(* PLC project canplc, CODESYS STW CODESYS V3.5 SP11 - ESX-3CS *)
(* stored: creationDateTime 2026-05-19T11:32:05.4310643, version 0.101, modificationDateTime 2026-02-01T07:40:15, organization Isoloader *)

TYPE t_can_errorfield : ARRAY[0..5] OF WORD;
END_TYPE

TYPE t_can_heartbeaterrors : ARRAY[0..7] OF BYTE;
END_TYPE

TYPE t_canopen_emcy : CIA405.EMCY_ERROR;
END_TYPE

TYPE t_node_state : _3SCOS.DEVICE_STATE;
END_TYPE

VAR_GLOBAL  (* GlobalVariablesCanplc *)
  gCANPLCBoolA : BOOL := TRUE;
END_VAR

FUNCTION_BLOCK CANOpenLocalDevice EXTENDS OperationalParticleSet
  VAR CONSTANT
    cHeartbeatTimer : t_time := TIME#500ms;
  END_VAR
  VAR
    lAlarmCANOpenMasterNotOperational : ReportableAlarmEscalating;
    lAlarmCANOpenMasterModulation : ReportableSignedModulation;
    lAlarmCANOpenMasterAllowableUp : ReportableAlarmAllowableUp;
    lVREnabled : ValueReferenceBool;
    lEnabled : BOOL := TRUE;
    lVRTriggerStart : ValueReferenceBool;
    lTriggerStart : BOOL := FALSE;
    lVROverrideConnected : ValueReferenceBool;
    lOverrideConnected : BOOL := FALSE;
    lModulationSystemStateScope : t_system_state;
    lOperationalSystemStateScope : t_system_state;
    lStartSystemStateScope : t_system_state;
    lModulationSeverity : t_severity;
    lNetworkId : BYTE;
    _EmergencyInfo : t_canopen_emcy;  (* foobar emcy messages not monitored *)
    lEmergencyInfo : REFERENCE TO t_canopen_emcy := _EmergencyInfo;
    lControllerId : BYTE := 0;
    lCANOpenDevice : REFERENCE TO _3SCSS.CANopenDevice;
    lMasterHeartbeat : HeartbeatHandler;
    lNodeState : t_node_state;
    lNodeStatePrev : t_node_state;
    lNMTStartCounter : USINT := 0;
    lNMTTimer : t_timer;
    lNMTEnableStart : BOOL := TRUE;
    lHeartbeatCounter : Counter;
    lHeartbeatTimer : t_timer;
    lEmergencyCounter : Counter;
    lReceiveEmcy : CIA405.RECV_EMCY_DEV;
    lEmergencyCode : WORD;
    lOverflowCounter : USINT := 0;
    lConnected : BOOL := TRUE;
  END_VAR

            ;
          

METHOD initialize
                  IF (NOT(__ISVALIDREF(lCANOpenDevice))) THEN
	gCodeErrorHandler(pMessage:=CONCAT('null reference in ',lIdentity));
END_IF

lAlarmCANOpenMasterNotOperational.initializeState(NopSelf,'',cACCANOpenMasterNotOperational);
lAlarmCANOpenMasterNotOperational.InitialSeverity := cSeverityWarning;
lAlarmCANOpenMasterNotOperational.SeverityWarningTimeout := T#0S;
lAlarmCANOpenMasterNotOperational.SeverityErrorTimeout := T#100MS;
lAlarmCANOpenMasterNotOperational.SeverityCriticalTimeout := T#5S;

lAlarmCANOpenMasterModulation.initializeState(NopSelf,'',cACCANOpenMasterModulation);
lAlarmCANOpenMasterModulation.pause(); // foobar - what impact does this have, should act as if not connected, ie put all joysticks to zero

lAlarmCANOpenMasterAllowableUp.initializeState(NopSelf,'',cACCANOpenMasterAllowableUp);
lAlarmCANOpenMasterAllowableUp.AllowableSystemState := cSystemStatePreOperational;
lAlarmCANOpenMasterAllowableUp.UpperSystemStateScope := cSystemStatePreOperational;
lAlarmCANOpenMasterAllowableUp.LowerSystemStateScope := cSystemStatePreOperational;
lAlarmCANOpenMasterAllowableUp.Life := 10;
lAlarmCANOpenMasterAllowableUp.InitialSeverity := cSeverityNone;
lAlarmCANOpenMasterAllowableUp.SeverityWarningTimeout := T#250MS;
lAlarmCANOpenMasterAllowableUp.SeverityErrorTimeout := T#1S;
lAlarmCANOpenMasterAllowableUp.SeverityCriticalTimeout := T#5S;	

lVREnabled.initializeValueReference(lEnabled,NopSelf,'Enabled','Enable canopen node','',cValueStyleParameter);
lVRTriggerStart.initializeValueReference(lTriggerStart,NopSelf,'TriggerStart','Trigger NMT message to take canopen node Operational','',cValueStyleTrigger);
lVROverrideConnected.initializeValueReference(lOverrideConnected,NopSelf,'OvrdConnected','Force state of canopen node to show as connected','',cValueStyleParameter);

SUPER^.initialize();
	
lModulationSystemStateScope := cSystemStateOperational;	
lOperationalSystemStateScope := cSystemStateGoOperational;
lStartSystemStateScope := cSystemStateGoOperational;
lModulationSeverity := cSeverityError;

lHeartbeatCounter.initialize();
lEmergencyCounter.initialize();
lMasterHeartbeat.initialize();

lHeartbeatTimer.initialize();
lHeartbeatTimer.Enable := TRUE;
lHeartbeatTimer.Period := cHeartbeatTimer;

lControllerId := lCANOpenDevice.NodeID;

lNMTStartCounter := 0;
lNMTTimer.Enable := TRUE;
lNMTTimer.Period := T#250MS;


                
END_METHOD

METHOD start
                  lCANOpenDevice.SwitchToOp();

lNMTStartCounter := lNMTStartCounter + 1;



                
END_METHOD

METHOD resetTraces : BOOL
                  lHeartbeatCounter.reset();
lEmergencyCounter.reset();
lOverflowCounter := 0;

lEmergencyInfo.EMCY_ERROR_CODE := 0;
lEmergencyInfo.ERROR_REGISTER := 0;
lEmergencyInfo.ERROR_FIELD[1] := 0;
lEmergencyInfo.ERROR_FIELD[2] := 0;
lEmergencyInfo.ERROR_FIELD[3] := 0;
lEmergencyInfo.ERROR_FIELD[4] := 0;
lEmergencyInfo.ERROR_FIELD[5] := 0;

                
END_METHOD

METHOD reset
                  
                
END_METHOD

METHOD emergencyHandler
  VAR_INPUT
    info : t_canopen_emcy;
  END_VAR
                  
                
END_METHOD

METHOD operator
                  SUPER^.operator();

IF (NOT(lEnabled)) THEN
	lNodeState := t_node_state.OPERATIONAL;
	lConnected := TRUE;
	RETURN;
END_IF

lNodeStatePrev := NodeState;
NodeState := LINT_TO_INT(INT_TO_LINT(lCANOpenDevice.State));

IF (((NodeState<>t_node_state.OPERATIONAL) AND (gSystemServices.SystemState.State>=lStartSystemStateScope)) OR
	(lTriggerStart)) THEN
	lTriggerStart := FALSE;
	start();
END_IF

lMasterHeartbeat.operator(); // foobar corrected - impact?
lHeartbeatCounter.operator();
lHeartbeatTimer.operator();

IF (lMasterHeartbeat.HeartbeatFault) THEN
	
	IF (gSystemServices.SystemState.State>=lOperationalSystemStateScope) THEN
		lAlarmCANOpenMasterNotOperational.trigger(FALSE);

		IF (lHeartbeatTimer.Expired) THEN
			lHeartbeatCounter.register();
		END_IF
	
		IF ((lAlarmCANOpenMasterNotOperational.Severity>=lModulationSeverity) AND
			(gSystemServices.SystemState.State>=lModulationSystemStateScope)) THEN
			lAlarmCANOpenMasterModulation.trigger(FALSE);
		END_IF
	END_IF
	
	lAlarmCANOpenMasterAllowableUp.test(FALSE);
ELSE
	lHeartbeatTimer.reset();
END_IF
lConnected := ((NOT(lHeartbeatTimer.Expired)) OR (lOverrideConnected)); // observational only

	
                
END_METHOD

METHOD initializeLocal
  VAR_INPUT
    device : REFERENCE TO _3SCSS.CANopenDevice;
    channel : USINT;
    handleHeartbeatHandler : UDINT;
  END_VAR
                  lCANOpenDevice REF= device;

lMasterHeartbeat.initializeMessage(handleHeartbeatHandler,channel);

                
END_METHOD

PROPERTY Operational : BOOL
GET
                    Operational := (NodeState=t_node_state.OPERATIONAL);
                  
END_GET
END_PROPERTY

PROPERTY EmergencyCounter : USINT
GET
                    EmergencyCounter := lEmergencyCounter.Count;
                  
END_GET
END_PROPERTY

PROPERTY OperationalSystemStateScope : t_system_state
GET
                    OperationalSystemStateScope := lOperationalSystemStateScope;
                  
END_GET
SET
                    lOperationalSystemStateScope := OperationalSystemStateScope;
                  
END_SET
END_PROPERTY

PROPERTY EmergencyInfo : t_canopen_emcy
GET
                    EmergencyInfo := lEmergencyInfo;
                  
END_GET
END_PROPERTY

PROPERTY HeartbeatCounter : USINT
GET
                    HeartbeatCounter := lHeartbeatCounter.Count;
                  
END_GET
END_PROPERTY

PROPERTY Connected : BOOL
GET
                    Connected := lConnected;


                  
END_GET
END_PROPERTY

PROPERTY OK : BOOL
GET
                    OK := ((NodeState=t_node_state.OPERATIONAL) OR
	(gSystemServices.SystemState.State<lOperationalSystemStateScope));

                  
END_GET
END_PROPERTY

PROPERTY NetworkId : BYTE
GET
                    NetworkId := lNetworkId;
                  
END_GET
SET
                    lNetworkId := NetworkId;
                  
END_SET
END_PROPERTY

PROPERTY EmergencyCode : WORD
GET
                    EmergencyCode := lEmergencyCode;
                  
END_GET
END_PROPERTY

PROPERTY ControllerId : BYTE
GET
                    ControllerId := lControllerId;

                  
END_GET
END_PROPERTY

PROPERTY Enabled : BOOL
GET
                    Enabled := lEnabled;
                  
END_GET
SET
                    lEnabled := Enabled;
                  
END_SET
END_PROPERTY

PROPERTY NodeState : t_node_state
GET
                    NodeState := lNodeState;
                  
END_GET
SET
                    lNodeState := NodeState;
                  
END_SET
END_PROPERTY

PROPERTY TypeToken : t_medium_string
GET
                    TypeToken := 'CANLocal';
                  
END_GET
END_PROPERTY
END_FUNCTION_BLOCK

FUNCTION_BLOCK CANOpenMaster EXTENDS OperationalParticleSet
  VAR
    lVREnable : ValueReferenceBool;
    lEnable : BOOL := TRUE;
    lAlarmChannelNotGood : ReportableAlarmAllowableUp;
    lAlarmChannelOperationalFail : ReportableSystemControl;
    lAlarmChannelNotOperational : ReportableAlarmEscalating;
    lAlarmChannelOverflow : ReportableAlarmEscalating;
    lAlarmChannelSlaveFailed : ReportableAlarmEscalating;
    lOperationalSystemStateScope : t_system_state;
    lAllowableUpSystemStateScope : t_system_state;
    lSystemControlRecovery : t_system_control;
    lBusPower : OutputSystemStateAuto;
    lEstopOnOverflow : BOOL := FALSE;
    lRestartOnOverflow : BOOL := FALSE;
    lEnablePerNodeHandling : BOOL := TRUE;
    lEstopOnNodeState : BOOL := FALSE;
    lRestartOnNodeState : BOOL := FALSE;
    lCANOpenManager : REFERENCE TO _3SCOS.CANopenManager;
    lGetDeviceState : CIA405.GET_STATE;
    lGetKernelState : CIA405.GET_CANOPEN_KERNEL_STATE;
    lChannelState : t_channel_state := cChannelStateNone;
    lMasterState : CIA405.DEVICE_STATE;
    lKernelState : CIA405.CANOPEN_KERNEL_ERROR;
    lKernel : _3SCOS.CANOPEN_KERNEL_STATE;
    lMandatoryBooted : BOOL;
    lOptionalBooted : BOOL;
    lClearErrors : BOOL;
    lClearRxOverflowFlag : BOOL;
    lClearTxOverflowFlag : BOOL;
    lRXOverflowFlag : BOOL;
    lTXOverflowFlag : BOOL;
    lHeartbeatErrorCount : UINT := 0;
    lTXOverflowErrorCount : UINT := 0;
    lRXOverflowErrorCount : UINT := 0;
    lResetCounter : USINT := 0;
    lNMT : CIA405.NMT;
    lNMTStartCounter : USINT := 0;
    lNMTStartAttemptCounter : USINT := 0;
    lNMTEnableStart : BOOL := FALSE;
    lTransmitNMT : TransmitNMT;
    lTransmitMessage : TransmitMessage;
  END_VAR

            ;
          

METHOD good
  VAR
    i : USINT;
  END_VAR
                  IF (lMasterState<>CIA405.DEVICE_STATE.OPERATIONAL) THEN
	lAlarmChannelNotOperational.trigger(FALSE);
	lChannelState := cChannelStateStarting;
	reset();
	RETURN;
END_IF

IF ((lEnablePerNodeHandling) AND (NOT(ChildrenOK))) THEN
	lAlarmChannelSlaveFailed.trigger(FALSE);

	IF (lRestartOnNodeState) THEN
		lChannelState := cChannelStateStarting;
		reset();
	END_IF
END_IF
                
END_METHOD

METHOD initialize
                  IF (NOT(__ISVALIDREF(lCANOpenManager))) THEN
	gCodeErrorHandler(pMessage:=CONCAT('null reference in ',lIdentity));
END_IF

lBusPower.Name := 'BusPower';
registerOperational(ADR(lBusPower));

lAlarmChannelNotGood.initializeState(NopSelf,'',cACChannelNotGood);
lAlarmChannelNotGood.AllowableSystemState := lAllowableUpSystemStateScope;
lAlarmChannelNotGood.UpperSystemStateScope := lAllowableUpSystemStateScope;
lAlarmChannelNotGood.LowerSystemStateScope := lAllowableUpSystemStateScope;
lAlarmChannelNotGood.InitialSeverity := cSeverityWarning;
lAlarmChannelNotGood.SeverityWarningTimeout := T#100MS;
lAlarmChannelNotGood.SeverityErrorTimeout := T#250MS;
lAlarmChannelNotGood.SeverityCriticalTimeout := T#2S;
lAlarmChannelNotGood.ForceTrigger := TRUE;

lAlarmChannelOperationalFail.initializeState(NopSelf,'',cACChannelOperationalFail);
lAlarmChannelOperationalFail.Control := lSystemControlRecovery;
lAlarmChannelOperationalFail.AllowableSystemState := lAllowableUpSystemStateScope;

lAlarmChannelNotOperational.initializeState(NopSelf,'',cACChannelNotOperational);
lAlarmChannelNotOperational.InitialSeverity := cSeverityWarning;
lAlarmChannelNotOperational.SeverityWarningTimeout := T#100MS;
lAlarmChannelNotOperational.SeverityErrorTimeout := T#250MS;
lAlarmChannelNotOperational.SeverityCriticalTimeout := T#1S;

lAlarmChannelOverflow.initializeState(NopSelf,'',cACChannelOverflow);
lAlarmChannelOverflow.InitialSeverity := cSeverityWarning;
lAlarmChannelOverflow.SeverityWarningTimeout := T#100MS;
lAlarmChannelOverflow.SeverityErrorTimeout := T#500MS;
lAlarmChannelOverflow.SeverityCriticalTimeout := T#1S;

lAlarmChannelSlaveFailed.initializeState(NopSelf,'',cACChannelSlaveFailed);
lAlarmChannelSlaveFailed.InitialSeverity := cSeverityWarning;
lAlarmChannelSlaveFailed.SeverityWarningTimeout := T#100MS;
lAlarmChannelSlaveFailed.SeverityErrorTimeout := T#1000MS;
lAlarmChannelSlaveFailed.SeverityCriticalTimeout := T#5S;

SUPER^.initialize();

lBusPower.OutputSystemState := cSystemStateStandby;

lChannelState := cChannelStateStarting;

lGetDeviceState.ENABLE := TRUE;
lGetDeviceState.DEVICE := 0;
lGetDeviceState.TIMEOUT := 200;

lGetKernelState.ENABLE := TRUE;
lGetKernelState.TIMEOUT := 200;

lNMT.DEVICE := 1;
lNMT.ENABLE := TRUE;
lNMT.TIMEOUT := 500;
lNMTStartCounter := 0;
lNMTStartAttemptCounter := 0;

lTransmitNMT.initialize();
lTransmitMessage.initialize();


                
END_METHOD

METHOD initializeMaster
  VAR_INPUT
    manager : REFERENCE TO _3SCOS.CANopenManager;
    channel : USINT;
    handleTransmitNMT : UDINT;
    handleTransmitMessage : UDINT;
  END_VAR
                  lCANOpenManager REF= manager;

lGetDeviceState.NETWORK := channel;
lGetKernelState.NETWORK := channel;
lNMT.NETWORK := channel;

lTransmitNMT.initializeMessage(handleTransmitNMT,channel);
lTransmitMessage.initializeMessage(handleTransmitMessage,channel);

                
END_METHOD

METHOD operator
  VAR
    i : USINT;
  END_VAR
                  IF (NOT(lEnable)) THEN
	lChannelState := cChannelStateGood;
	RETURN;
END_IF

SUPER^.operator();

CASE lChannelState OF
	cChannelStateNone:
		;
	cChannelStateError:
		starting();
	cChannelStateStarting:
		starting();
	cChannelStateGood:
		good();
	cChannelStateOverflow:
		starting();
	cChannelStateHeartbeat:
		starting();
	cChannelStateEmergency:
		starting();
END_CASE

lKernel := lCANOpenManager.KernelState;
lMandatoryBooted := lCANOpenManager.MandatorySlavesBooted;
lOptionalBooted := lCANOpenManager.OptionalSlavesBooted;

lGetDeviceState.ENABLE := TRUE;
lGetDeviceState();
IF (lGetDeviceState.CONFIRM) THEN
	lMasterState := lGetDeviceState.STATE;
END_IF
IF ((lGetDeviceState.CONFIRM) OR (lGetDeviceState.ERROR<>CIA405.CANOPEN_KERNEL_ERROR.CANOPEN_KERNEL_NO_ERROR)) THEN
	lGetDeviceState.ENABLE := FALSE;
	lGetDeviceState();
END_IF

lGetKernelState.ENABLE := TRUE;
lGetKernelState();
IF (lGetKernelState.CONFIRM) THEN
	lKernelState := lGetKernelState.STATE;
END_IF
IF ((lGetKernelState.CONFIRM) OR (lGetKernelState.ERROR<>CIA405.CANOPEN_KERNEL_ERROR.CANOPEN_KERNEL_NO_ERROR)) THEN
	lGetKernelState.ENABLE := FALSE;
	lGetKernelState();
END_IF

IF (lChannelState<cChannelStateGood) THEN
	lAlarmChannelNotGood.trigger(FALSE);
	
	IF (gSystemServices.SystemState.State>=lOperationalSystemStateScope) THEN
		lAlarmChannelOperationalFail.trigger(FALSE);
	END_IF
END_IF

CASE lKernelState OF
	CIA405.CANOPEN_KERNEL_ERROR.CANOPEN_KERNEL_DATA_OVERFLOW:
		overflow();
END_CASE

                
END_METHOD

METHOD overflow
                  lAlarmChannelOverflow.report(FALSE);

IF ((lEstopOnOverflow) AND (gSystemServices.SystemState.State=cSystemStateOperational)) THEN
	lAlarmChannelOverflow.propagate(); //foobar should be pause everything due to canbus system health, or go slow on all travel
END_IF

IF (lRestartOnOverflow) THEN
	lChannelState := cChannelStateStarting;
	reset();
END_IF


                
END_METHOD

METHOD reset
                  lResetCounter := lResetCounter + 1;
                
END_METHOD

METHOD restart
                  lNMT.STATE := CIA405.TRANSITION_STATE.RESET_NODE;
lNMT.DEVICE := 1;
lNMT.ENABLE := lNMTEnableStart;
lNMT();
IF ((lNMT.CONFIRM) OR (lNMT.ERROR<>CIA405.CANOPEN_KERNEL_ERROR.CANOPEN_KERNEL_NO_ERROR)) THEN
	lNMT.ENABLE := FALSE;
	lNMTStartAttemptCounter := lNMTStartAttemptCounter + 1;
	IF (lNMT.CONFIRM) THEN
		lNMTStartCounter := lNMTStartCounter + 1;
	END_IF
	lNMT();
END_IF
                
END_METHOD

METHOD starting
                  IF (lMasterState=CIA405.DEVICE_STATE.OPERATIONAL) THEN
	lChannelState := cChannelStateGood;
END_IF
                
END_METHOD

METHOD initializeMasterPower
  VAR_INPUT
    busPower : REFERENCE TO DINT;
  END_VAR
                  lBusPower.OutputObject.OutputReference REF= busPower;

                
END_METHOD

PROPERTY BusPower : BOOL
GET
                    BusPower := lBusPower.State;
                  
END_GET
END_PROPERTY

PROPERTY ChannelState : t_channel_state
GET
                    ChannelState := lChannelState;
                  
END_GET
END_PROPERTY

PROPERTY MasterState : CIA405.DEVICE_STATE
GET
                    MasterState := lMasterState;
                  
END_GET
END_PROPERTY

PROPERTY TransmitMessage : REFERENCE TO TransmitMessage
GET
                    TransmitMessage ref= lTransmitMessage;
                  
END_GET
END_PROPERTY

PROPERTY TransmitNMT : REFERENCE TO TransmitNMT
GET
                    TransmitNMT ref= lTransmitNMT;
                  
END_GET
END_PROPERTY

PROPERTY TypeToken : t_medium_string
GET
                    TypeToken := 'CANMaster';
                  
END_GET
END_PROPERTY
END_FUNCTION_BLOCK

FUNCTION_BLOCK CANOpenSlave EXTENDS OperationalParticleSet
  VAR_INPUT
    lAlarmCANOpenSlaveModulation : ReportableSignedModulation;
  END_VAR
  VAR CONSTANT
    cNodeStatePeriod : t_time := TIME#10ms;
    cHeartbeatPeriod : t_time := TIME#50ms;
    cEmergencyRegisterMax : USINT := 16;
  END_VAR
  VAR
    lAlarmCANOpenSlaveNotOperational : ReportableAlarmEscalating;
    lAlarmCANOpenSlaveAllowableUp : ReportableAlarmAllowableUp;
    lAlarmCANOpenSlaveNotify : ReportableAlarm;
    lAlarmCANOpenSlaveBlock : LockoutInterlock;
    lAlarmCANOpenSlaveStop : ReportableSystemControl;
    lVREnabled : ValueReferenceBool;
    lEnabled : BOOL := TRUE;
    lVRTriggerStart : ValueReferenceBool;
    lTriggerStart : BOOL := FALSE;
    lVROverrideConnected : ValueReferenceBool;
    lOverrideConnected : BOOL := FALSE;
    lModulationSystemStateScope : t_system_state;
    lOperationalSystemStateScopeLower : t_system_state;
    lOperationalSystemStateScopeUpper : t_system_state;
    lStartSystemStateScope : t_system_state;
    lModulationSeverity : t_severity;
    lNetworkId : BYTE;
    _EmergencyInfo : t_canopen_emcy;
    lEmergencyInfo : REFERENCE TO t_canopen_emcy := _EmergencyInfo;
    lControllerId : BYTE := 0;
    lCANRemoteDevice : REFERENCE TO _3SCOS.CANRemoteDevice;
    lMaster : REFERENCE TO CANOpenMaster;
    lNodeState : t_node_state;
    lNodeStatePrev : t_node_state;
    lNMTStartCounter : USINT := 0;
    lNMTTimer : t_timer;
    lNMTEnableStart : BOOL := TRUE;
    lHeartbeatCounter : Counter;
    lHeartbeatTimer : t_timer;
    lNodeStateTimer : t_timer;
    lEmergencyCounter : Counter;
    lEmergencyClearCount : USINT := 0;
    lReceiveEmcy : CIA405.RECV_EMCY_DEV;
    lEmergencyCode : WORD;
    lSDOWrite : CIA405.SDO_WRITE_DATA;
    lSDOWriteData : DWORD;
    lSDOWriteAttemptCounter : USINT := 0;
    lSDOWriteSuccessCounter : USINT := 0;
    lSDORead : CIA405.SDO_READ_DATA;
    lSDOReadData : DWORD;
    lSDOLastSuccessfulReadData : DWORD;
    lSDODReadDataLength : UDINT := 4;
    lSDOReadSuccess : BOOL := FALSE;
    lSDOReadAttemptCounter : USINT := 0;
    lSDOReadSuccessCounter : USINT := 0;
    lOverflowCounter : USINT := 0;
    lStartHandlerCounter : UINT := 0;
    lConnected : BOOL := TRUE;
    lEmergencyRegister : ARRAY[1..cEmergencyRegisterMax] OF t_canopen_emcy;
    lEmergencyCount : USINT := 0;
  END_VAR

            ;
          

METHOD cancelSDORead
                  lSDORead.ENABLE := FALSE;
lSDODReadDataLength := 4;
lSDORead(DATALENGTH:=lSDODReadDataLength);

                
END_METHOD

METHOD cancelSDOWrite
                  lSDOWrite.ENABLE := FALSE;
lSDOWrite();
                
END_METHOD

METHOD emergencyHandler
  VAR_INPUT
    info : t_canopen_emcy;
  END_VAR
                  emergencyRegisterAdd(info);
lAlarmCANOpenSlaveNotify.triggerWithContext(WORD_TO_LWORD(info.EMCY_ERROR_CODE));



                
END_METHOD

METHOD initialize
                  IF ((NOT(__ISVALIDREF(lCANRemoteDevice))) OR
	(NOT(__ISVALIDREF(lMaster)))) THEN
	gCodeErrorHandler(pMessage:=CONCAT('null reference in ',lIdentity));
END_IF

lAlarmCANOpenSlaveNotOperational.initializeState(NopSelf,'',cACCANOpenSlaveNotOperational);
lAlarmCANOpenSlaveNotOperational.InitialSeverity := cSeverityWarning;
lAlarmCANOpenSlaveNotOperational.SeverityWarningTimeout := T#0S;
lAlarmCANOpenSlaveNotOperational.SeverityErrorTimeout := T#100MS;
lAlarmCANOpenSlaveNotOperational.SeverityCriticalTimeout := T#5S;

lAlarmCANOpenSlaveModulation.initializeState(NopSelf,'',cACCANOpenSlaveModulation); // foobar life was zero
lAlarmCANOpenSlaveModulation.pause();

lAlarmCANOpenSlaveAllowableUp.initializeState(NopSelf,'',cACCANOpenSlaveAllowableUp);
lAlarmCANOpenSlaveAllowableUp.AllowableSystemState := cSystemStateGoOperational;
lAlarmCANOpenSlaveAllowableUp.UpperSystemStateScope := cSystemStateGoOperational;
lAlarmCANOpenSlaveAllowableUp.LowerSystemStateScope := cSystemStateGoOperational;
lAlarmCANOpenSlaveAllowableUp.Life := 10;
lAlarmCANOpenSlaveAllowableUp.InitialSeverity := cSeverityNone;
lAlarmCANOpenSlaveAllowableUp.SeverityWarningTimeout := T#250MS;
lAlarmCANOpenSlaveAllowableUp.SeverityErrorTimeout := T#1S;
lAlarmCANOpenSlaveAllowableUp.SeverityCriticalTimeout := T#5S;	

lVREnabled.initializeValueReference(lEnabled,NopSelf,'Enabled','Enable canopen node','',cValueStyleParameter);
lVRTriggerStart.initializeValueReference(lTriggerStart,NopSelf,'TriggerStart','Trigger NMT message to take canopen node Operational','',cValueStyleTrigger);
lVROverrideConnected.initializeValueReference(lOverrideConnected,NopSelf,'OvrdConnected','Force state of canopen node to show as connected','',cValueStyleParameter);

lAlarmCANOpenSlaveNotify.initializeState(NopSelf,'',cACCANOpenSlaveNotify);
lAlarmCANOpenSlaveNotify.Life := 10;
lAlarmCANOpenSlaveNotify.Severity := cSeverityWarning;

lAlarmCANOpenSlaveBlock.initializeState(NopSelf,'',cACCANOpenSlaveBlock);
lAlarmCANOpenSlaveBlock.Life := 10;

lAlarmCANOpenSlaveStop.initializeState(NopSelf,'',cACCANOpenSlaveStop); // foobar life was zero
lAlarmCANOpenSlaveStop.Control := cSystemControlStop; //foobar consider restart
lAlarmCANOpenSlaveStop.AllowableSystemState := cSystemStatePreOperational;

SUPER^.initialize();

lModulationSystemStateScope := cSystemStateOperational;	
lOperationalSystemStateScopeLower := cSystemStateOperational;
lOperationalSystemStateScopeUpper := cSystemStateOperational;
lStartSystemStateScope := cSystemStateGoOperational;
lModulationSeverity := cSeverityError;

lHeartbeatCounter.initialize();
lEmergencyCounter.initialize();

lHeartbeatTimer.initialize();
lHeartbeatTimer.Enable := TRUE;
lHeartbeatTimer.Period := cHeartbeatPeriod;

lNodeStateTimer.initialize();
lNodeStateTimer.Enable := TRUE;
lNodeStateTimer.Period := cNodeStatePeriod;

lCANRemoteDevice.NMTErrorBehaviour := _3SCOS.NMT_ERROR_BEHAVIOUR.RESTART_SLAVE;
lControllerId := lCANRemoteDevice.NodeID;

//lNMT.DEVICE := lControllerId;
//lNMT.ENABLE := TRUE;
//lNMT.NETWORK := lNetworkId;
//lNMT.TIMEOUT := 500;
lNMTStartCounter := 0;
lNMTTimer.Enable := TRUE;
lNMTTimer.Period := T#250MS;
//lNMTStartFailedCounter := 0;

lSDOWrite.DEVICE := lControllerId;
lSDOWrite.CHANNEL := 0;
lSDOWrite.NETWORK := lNetworkId;
lSDOWrite.ENABLE := FALSE;
lSDOWrite.TIMEOUT := 500;
lSDOWrite.MODE := CIA405.SDO_MODE.AUTO;
lSDOWrite.DATA := ADR(lSDOWriteData);

lSDORead.DEVICE := lControllerId;
lSDORead.CHANNEL := 0;
lSDORead.NETWORK := lNetworkId;
lSDORead.ENABLE := FALSE;
lSDORead.TIMEOUT := 500;
lSDORead.MODE := CIA405.SDO_MODE.AUTO;
lSDORead.DATA := ADR(lSDOReadData);

lReceiveEmcy.DEVICE := lControllerId;
lReceiveEmcy.ENABLE := TRUE;
lReceiveEmcy.NETWORK := lNetworkId;
lReceiveEmcy.TIMEOUT := 200;

                
END_METHOD

METHOD initializeSlave
  VAR_INPUT
    device : REFERENCE TO _3SCOS.CANRemoteDevice;
    master : REFERENCE TO CANOpenMaster;
  END_VAR
                  lCANRemoteDevice REF= device;
lMaster REF= master;


                
END_METHOD

METHOD operator
                  SUPER^.operator();

IF (NOT(lEnabled)) THEN
	lNodeState := t_node_state.OPERATIONAL;
	lConnected := TRUE;
	RETURN;
END_IF

lNodeStatePrev := NodeState;
NodeState := lCANRemoteDevice.CANopenState;

IF (((NodeState=t_node_state.PRE_OPERATIONAL) AND (gSystemServices.SystemState.State>=lStartSystemStateScope)) OR
	(lTriggerStart)) THEN
	lTriggerStart := FALSE;
	start();
END_IF

IF ((gSystemServices.SystemState.State>=lStartSystemStateScope) AND (gSystemServices.SystemState.State<lOperationalSystemStateScopeLower)) THEN
	startHandler();
END_IF

IF (gSystemServices.SystemState.State<lStartSystemStateScope) THEN
	startResetHandler();
END_IF

IF (lSDOWrite.ENABLE) THEN
	lSDOWrite();
	IF ((lSDOWrite.CONFIRM) OR (lSDOWrite.ERROR<>CIA405.CANOPEN_KERNEL_ERROR.CANOPEN_KERNEL_NO_ERROR)) THEN
		lSDOWrite.ENABLE := FALSE;
		lSDOWriteAttemptCounter := lSDOWriteAttemptCounter + 1;
		IF (lSDOWrite.CONFIRM) THEN
			lSDOWriteSuccessCounter := lSDOWriteSuccessCounter + 1;
		END_IF
	END_IF	
END_IF

IF (lSDORead.ENABLE) THEN
	lSDORead(DATALENGTH:=lSDODReadDataLength);
	IF ((lSDORead.CONFIRM) OR (lSDORead.ERROR<>CIA405.CANOPEN_KERNEL_ERROR.CANOPEN_KERNEL_NO_ERROR)) THEN
		lSDORead.ENABLE := FALSE;
		lSDOReadAttemptCounter := lSDOReadAttemptCounter + 1;
		IF (lSDORead.CONFIRM) THEN
			lSDOReadSuccess := TRUE;
			sdoReadHandler();
			lSDOLastSuccessfulReadData := lSDOReadData;
			lSDOReadSuccessCounter := lSDOReadSuccessCounter + 1;
		END_IF
	END_IF	
END_IF

lHeartbeatCounter.operator();
lHeartbeatTimer.operator();

IF (NodeState<>t_node_state.OPERATIONAL) THEN
	
	notOperational();
	
	IF ((gSystemServices.SystemState.State>=lOperationalSystemStateScopeLower) AND
		(gSystemServices.SystemState.State<=lOperationalSystemStateScopeUpper)) THEN
		lAlarmCANOpenSlaveNotOperational.trigger(FALSE);

		IF ((NodeState=t_node_state.NOT_AVAIL) AND 
			(lHeartbeatTimer.Expired)) THEN
			lHeartbeatCounter.register();
		END_IF
	
		IF ((lAlarmCANOpenSlaveNotOperational.Severity>=lModulationSeverity) AND
			(gSystemServices.SystemState.State>=lModulationSystemStateScope)) THEN
			lAlarmCANOpenSlaveModulation.trigger(FALSE);
		END_IF
	END_IF
	
	lAlarmCANOpenSlaveAllowableUp.test(FALSE);
ELSE
	lHeartbeatTimer.reset();
END_IF
lConnected := ((NOT(lHeartbeatTimer.Expired)) OR (lOverrideConnected)); // observational only

lReceiveEmcy.ENABLE := TRUE;
lReceiveEmcy();
IF (lReceiveEmcy.CONFIRM) THEN
	lEmergencyCounter.operator();
	
	IF (lReceiveEmcy.ERRORINFO.EMCY_ERROR_CODE<>0) THEN
		lEmergencyCounter.register();
		lEmergencyInfo := lReceiveEmcy.ERRORINFO;
		IF (gCANPLCBoolA) THEN emergencyHandler(lReceiveEmcy.ERRORINFO); END_IF
	ELSE
		emergencyRegisterClear();
	END_IF
	
	lEmergencyCode := lReceiveEmcy.ERRORINFO.EMCY_ERROR_CODE;
END_IF
IF ((lReceiveEmcy.CONFIRM) OR (lReceiveEmcy.ERROR<>CIA405.CANOPEN_KERNEL_ERROR.CANOPEN_KERNEL_NO_ERROR)) THEN
	lReceiveEmcy.ENABLE := FALSE;
	lReceiveEmcy();
END_IF

                
END_METHOD

METHOD requestSDORead : BOOL
  VAR_INPUT
    force : BOOL;
    index : WORD;
    subindex : BYTE;
    length : UDINT;
  END_VAR
                  IF (force) THEN
	cancelSDORead();
END_IF

IF (lSDORead.ENABLE) THEN
	requestSDORead := FALSE;
	RETURN;
END_IF

requestSDORead := TRUE;

lSDORead.ENABLE := TRUE;

lSDORead.INDEX := index;
lSDORead.SUBINDEX := subindex;
lSDODReadDataLength := length;

lSDOReadSuccess := FALSE;

                
END_METHOD

METHOD requestSDOWrite : BOOL
  VAR_INPUT
    force : BOOL;
    index : WORD;
    subindex : BYTE;
    data : DWORD;
    length : UDINT;
  END_VAR
                  IF (force) THEN
	cancelSDOWrite();
END_IF

IF (lSDOWrite.ENABLE) THEN
	requestSDOWrite := FALSE;
	RETURN;
END_IF

requestSDOWrite := FALSE;

lSDOWrite.ENABLE := TRUE;

lSDOWrite.INDEX := index;
lSDOWrite.SUBINDEX := subindex;
lSDOWrite.DATALENGTH := length;

lSDOWriteData := data;


                
END_METHOD

METHOD reset
                  
                
END_METHOD

METHOD sdoReadHandler
                  ;
                
END_METHOD

METHOD start
                  lNMTTimer.operator();
IF (lNMTTimer.Expired) THEN
	lMaster.TransmitNMT.startNode(lControllerId);
	lNMTStartCounter := lNMTStartCounter + 1;
	lNMTTimer.reset();
END_IF

(*lNMT.STATE := CIA405.TRANSITION_STATE.START_REMOTE_NODE;
IF (lNMTStartFailedCounter>5) THEN
	lNMT.STATE := CIA405.TRANSITION_STATE.STOP_REMOTE_NODE;
END_IF
IF (lNMTStartFailedCounter>10) THEN
	lNMT.STATE := CIA405.TRANSITION_STATE.RESET_NODE;
END_IF
IF (lNMTStartFailedCounter>15) THEN
	lNMT.STATE := CIA405.TRANSITION_STATE.RESET_COMMUNICATION;
END_IF
IF (lNMTStartFailedCounter>20) THEN
	lMaster.restart();
END_IF

lNMT.DEVICE := lControllerId;
lNMT.ENABLE := lNMTEnableStart;
lNMT();
IF ((lNMT.CONFIRM) OR (lNMT.ERROR<>CIA405.CANOPEN_KERNEL_ERROR.CANOPEN_KERNEL_NO_ERROR)) THEN
	lNMT.ENABLE := FALSE;
	IF (lNMT.CONFIRM) THEN
		lNMTStartCounter := lNMTStartCounter + 1;
		lNMTStartFailedCounter := 0;
	ELSE
		lNMTStartFailedCounter := lNMTStartFailedCounter + 1;
	END_IF
	lNMT();
END_IF
*)

                
END_METHOD

METHOD startHandler
                  lStartHandlerCounter := lStartHandlerCounter + 1;
                
END_METHOD

METHOD startResetHandler
                  ;
                
END_METHOD

METHOD emergencyRegisterAdd : BOOL
  VAR_INPUT
    info : t_canopen_emcy;
  END_VAR
  VAR
    i : USINT;
  END_VAR
                  emergencyRegisterAdd := FALSE;

IF (info.EMCY_ERROR_CODE=0) THEN
	RETURN;
END_IF

FOR i:=1 TO lEmergencyCount DO
	IF (lEmergencyRegister[i].EMCY_ERROR_CODE=info.EMCY_ERROR_CODE) THEN
		RETURN;
	END_IF
END_FOR

IF (lEmergencyCount>=cEmergencyRegisterMax) THEN
	gConfigErrorHandler(pMessage:=CONCAT('overflow in emergency register in',lIdentity));
	RETURN;
END_IF

lEmergencyCount := lEmergencyCount + 1;
lEmergencyRegister[lEmergencyCount] := info;
emergencyRegisterAdd := TRUE;

                
END_METHOD

METHOD describe
  VAR_INPUT
    executeContext : POINTER TO ExecuteContext;
  END_VAR
  VAR
    i : UINT;
    str : t_stream_string;
  END_VAR
                  SUPER^.describe(executeContext);

executeContext^.appendPair('node',BYTE_TO_STRING(lControllerId),FALSE,TRUE);

IF (executeContext^.matchOption(cExecuteOptionVerbose)) THEN
	executeContext^.append('"current_emcy": ');
	executeContext^.recordInitiator();
		
	executeContext^.appendPair('code',WORD_TO_STRING(lEmergencyRegister[i].EMCY_ERROR_CODE),FALSE,FALSE);
	executeContext^.appendPair('register',BYTE_TO_STRING(lEmergencyRegister[i].ERROR_REGISTER),FALSE,TRUE);
	executeContext^.appendPair('field_1',BYTE_TO_STRING(lEmergencyRegister[i].ERROR_FIELD[1]),FALSE,TRUE);
	executeContext^.appendPair('field_2',BYTE_TO_STRING(lEmergencyRegister[i].ERROR_FIELD[2]),FALSE,TRUE);
	executeContext^.appendPair('field_3',BYTE_TO_STRING(lEmergencyRegister[i].ERROR_FIELD[3]),FALSE,TRUE);
	executeContext^.appendPair('field_4',BYTE_TO_STRING(lEmergencyRegister[i].ERROR_FIELD[4]),FALSE,TRUE);
	executeContext^.appendPair('field_5',BYTE_TO_STRING(lEmergencyRegister[i].ERROR_FIELD[5]),FALSE,TRUE);

	executeContext^.recordTerminator();
END_IF

                
END_METHOD

METHOD emergencyRegisterClear
                  lEmergencyCount := 0;
lEmergencyClearCount := lEmergencyClearCount + 1;

                
END_METHOD

METHOD notOperational
                  
                
END_METHOD

PROPERTY Connected : BOOL
GET
                    Connected := lConnected;

                  
END_GET
END_PROPERTY

PROPERTY ControllerId : BYTE
GET
                    ControllerId := lControllerId;

                  
END_GET
END_PROPERTY

PROPERTY EmergencyCode : WORD
GET
                    EmergencyCode := lEmergencyCode;
                  
END_GET
END_PROPERTY

PROPERTY EmergencyCounter : USINT
GET
                    EmergencyCounter := lEmergencyCounter.Count;
                  
END_GET
END_PROPERTY

PROPERTY EmergencyInfo : t_canopen_emcy
GET
                    EmergencyInfo := lEmergencyInfo;
                  
END_GET
END_PROPERTY

PROPERTY Enabled : BOOL
GET
                    Enabled := lEnabled;
                  
END_GET
SET
                    lEnabled := Enabled;
                  
END_SET
END_PROPERTY

PROPERTY HealthSystemStateScope : t_system_state
GET
                    HealthSystemStateScope := lModulationSystemStateScope;
                  
END_GET
SET
                    lModulationSystemStateScope := HealthSystemStateScope;
                  
END_SET
END_PROPERTY

PROPERTY HeartbeatCounter : USINT
GET
                    HeartbeatCounter := lHeartbeatCounter.Count;
                  
END_GET
END_PROPERTY

PROPERTY NetworkId : BYTE
GET
                    NetworkId := lNetworkId;
                  
END_GET
SET
                    lNetworkId := NetworkId;
                  
END_SET
END_PROPERTY

PROPERTY NodeState : t_node_state
GET
                    NodeState := lNodeState;
                  
END_GET
SET
                    IF (NodeState=t_node_state.OPERATIONAL) THEN
	lNodeStateTimer.reset();
	lNodeState := NodeState;
	RETURN;
END_IF

lNodeStateTimer.operator();

IF ((lNodeState=t_node_state.OPERATIONAL) AND
	(NOT(lNodeStateTimer.Expired))) THEN
	RETURN;
END_IF

lNodeState := NodeState;

                  
END_SET
END_PROPERTY

PROPERTY OK : BOOL
GET
                    OK := ((NodeState=t_node_state.OPERATIONAL) OR
	(gSystemServices.SystemState.State<lOperationalSystemStateScopeLower) OR
	(gSystemServices.SystemState.State>lOperationalSystemStateScopeUpper));

                  
END_GET
END_PROPERTY

PROPERTY Operational : BOOL
GET
                    Operational := (NodeState=t_node_state.OPERATIONAL);
                  
END_GET
END_PROPERTY

PROPERTY OperationalSystemStateScopeLower : t_system_state
GET
                    OperationalSystemStateScopeLower := lOperationalSystemStateScopeLower;
                  
END_GET
SET
                    lOperationalSystemStateScopeLower := OperationalSystemStateScopeLower;
                  
END_SET
END_PROPERTY

PROPERTY OverflowCounter : USINT
GET
                    OverflowCounter := lOverflowCounter;
                  
END_GET
END_PROPERTY

PROPERTY TypeToken : t_medium_string
GET
                    TypeToken := 'CANSlave';
                  
END_GET
END_PROPERTY

PROPERTY OperationalSystemStateScopeUpper : t_system_state
GET
                    OperationalSystemStateScopeUpper := lOperationalSystemStateScopeUpper;
                  
END_GET
SET
                    lOperationalSystemStateScopeUpper := OperationalSystemStateScopeUpper;
                  
END_SET
END_PROPERTY
END_FUNCTION_BLOCK

FUNCTION_BLOCK SDOReadCANMessage EXTENDS CANMessage
  VAR
    lSDORead : CIA405.SDO_READ_DATA;
    lSDOReadData : DWORD;
    lSDODReadDataLength : UDINT;
    lSDOReadAttemptCounter : USINT := 0;  (* lSDOLastSuccessfulReadData: DWORD; *)
    lSDOReadSuccessCounter : USINT := 0;
    lProceedOnFail : BOOL := TRUE;
    lProceedOnOverflow : BOOL := TRUE;
  END_VAR

            
          

METHOD cancelSDORead
                  lSDORead.ENABLE := FALSE;
lSDORead(DATALENGTH:=lSDODReadDataLength);

                
END_METHOD

METHOD initialize
                  SUPER^.initialize();

lSDOReadAttemptCounter := 0;
lSDOReadSuccessCounter := 0;

lSDORead.CHANNEL := 0;
lSDORead.ENABLE := FALSE;
lSDORead.TIMEOUT := 500;
lSDORead.MODE := CIA405.SDO_MODE.AUTO;
lSDORead.DATA := ADR(lSDOReadData);
                
END_METHOD

METHOD operator
                  SUPER^.operator();

IF (lSDORead.ENABLE) THEN
	lSDORead(DATALENGTH:=lSDODReadDataLength);
	IF ((lSDORead.CONFIRM) OR (lSDORead.ERROR<>CIA405.CANOPEN_KERNEL_ERROR.CANOPEN_KERNEL_NO_ERROR)) THEN
		lSDORead.ENABLE := FALSE;
		lSDOReadAttemptCounter := lSDOReadAttemptCounter + 1;
		IF (lSDORead.CONFIRM) THEN
			lSuccess := TRUE;
			lFinished := TRUE;
			lProceed := TRUE;
			
			sdoReadHandler();
			lSDOReadSuccessCounter := lSDOReadSuccessCounter + 1;
			
			finish();
			RETURN;
		END_IF
		IF (lSDORead.ERROR<>CIA405.CANOPEN_KERNEL_ERROR.CANOPEN_KERNEL_NO_ERROR) THEN
			lSuccess := FALSE;
			lFinished := TRUE;
			lProceed := TRUE;
			
			finish();
			RETURN;
		END_IF
	END_IF	
END_IF

                
END_METHOD

METHOD reset
                  SUPER^.reset();
                
END_METHOD

METHOD sdoReadHandler
                  ;
                
END_METHOD

METHOD start
                  cancelSDORead();
lSDORead.ENABLE := TRUE;

SUPER^.start();
                
END_METHOD

PROPERTY ControllerId : BYTE
GET
                    ControllerId := lSDORead.DEVICE;

                  
END_GET
SET
                    lSDORead.DEVICE := ControllerId;
                  
END_SET
END_PROPERTY

PROPERTY NetworkId : BYTE
GET
                    NetworkId := lSDORead.NETWORK;

                  
END_GET
SET
                    lSDORead.NETWORK := NetworkId;
                  
END_SET
END_PROPERTY
END_FUNCTION_BLOCK

FUNCTION_BLOCK SDOWriteCANMessage EXTENDS CANMessage
  VAR
    lSDOWrite : CIA405.SDO_WRITE_DATA;
    lSDOWriteData : DWORD;
    lSDOWriteAttemptCounter : USINT := 0;
    lSDOWriteSuccessCounter : USINT := 0;
    lProceedOnFail : BOOL := TRUE;
    lProceedOnOverflow : BOOL := TRUE;
  END_VAR

            
          

METHOD cancelSDOWrite
                  lSDOWrite.ENABLE := FALSE;
lSDOWrite();
                
END_METHOD

METHOD initialize
                  SUPER^.initialize();

lSDOWriteAttemptCounter := 0;
lSDOWriteSuccessCounter := 0;

lSDOWrite.CHANNEL := 0;
lSDOWrite.ENABLE := FALSE;
lSDOWrite.TIMEOUT := 500;
lSDOWrite.MODE := CIA405.SDO_MODE.AUTO;
lSDOWrite.DATA := ADR(lSDOWriteData);
                
END_METHOD

METHOD operator
                  SUPER^.operator();

IF (lSDOWrite.ENABLE) THEN
	lSDOWrite();
	IF ((lSDOWrite.CONFIRM) OR (lSDOWrite.ERROR<>CIA405.CANOPEN_KERNEL_ERROR.CANOPEN_KERNEL_NO_ERROR)) THEN
		lSDOWrite.ENABLE := FALSE;
		lSDOWriteAttemptCounter := lSDOWriteAttemptCounter + 1;
		IF (lSDOWrite.CONFIRM) THEN
			lSuccess := TRUE;
			lFinished := TRUE;
			lProceed := TRUE;
			
			lSDOWriteSuccessCounter := lSDOWriteSuccessCounter + 1;
			
			finish();
			RETURN;
		END_IF
		IF (lSDOWrite.ERROR<>CIA405.CANOPEN_KERNEL_ERROR.CANOPEN_KERNEL_NO_ERROR) THEN
			lSuccess := FALSE;
			lFinished := TRUE;
			lProceed := TRUE;
			
			finish();
			RETURN;
		END_IF
	END_IF	
END_IF


                
END_METHOD

METHOD reset
                  SUPER^.reset();
                
END_METHOD

METHOD start
                  cancelSDOWrite();
lSDOWrite.ENABLE := TRUE;

SUPER^.start();
                
END_METHOD

PROPERTY ControllerId : BYTE
GET
                    ControllerId := lSDOWrite.DEVICE;

                  
END_GET
SET
                    lSDOWrite.DEVICE := ControllerId;
                  
END_SET
END_PROPERTY

PROPERTY NetworkId : BYTE
GET
                    NetworkId := lSDOWrite.NETWORK;

                  
END_GET
SET
                    lSDOWrite.NETWORK := NetworkId;
                  
END_SET
END_PROPERTY
END_FUNCTION_BLOCK

FUNCTION_BLOCK MimicCANOpenSlave EXTENDS CANOpenSlave

            ;
          

METHOD initialize
                  SUPER^.initialize();

lNodeStateTimer.Period := T#2S;

                
END_METHOD

PROPERTY TypeToken : t_medium_string
GET
                    TypeToken := 'MimicCANSlave';
                  
END_GET
END_PROPERTY
END_FUNCTION_BLOCK

FUNCTION_BLOCK ControllerSecondaryPowerSupply EXTENDS MimicCANOpenSlave
  VAR CONSTANT
    cAvailabilityTemperatureWarning : t_percentage := 0.5;
    cAvailabilityTemperatureFault : t_percentage := 0.25;
  END_VAR
  VAR_GLOBAL
    sControllerSecondaryPowerSupply : t_medium_string := 'cSecondary';
  END_VAR
  VAR
    lRequestedRunState : ValueObjectEnumTypeOutputReferenceUSINT;
    lTargetVoltage : ValueObjectRealScaledOffsetOutputReferenceUSINT;
    lVoltage : ValueObjectRealScaledOffsetInputReferenceUINTSwitched;
    lCurrent : ValueObjectRealScaledOffsetInputReferenceUINTSwitched;
    lTemperature : ValueObjectRealScaledOffsetInputReferenceUSINT;
    lDiagnosticState : ValueObjectUINTInputReferenceUINT;
    lStatusInitialization : ValueObjectBoolInputReferenceUINT;
    lStatusWorking : ValueObjectBoolInputReferenceUINT;
    lAlarmSecondaryTemperature : ReportableSignedModulation;
    lCurrentRunState : ValueObjectEnumType;
    lSecondaryPowerSupply : REFERENCE TO SecondaryPowerSupply;
  END_VAR

            ;
          

METHOD initialize
                  IF (NOT(__ISVALIDREF(lSecondaryPowerSupply))) THEN
	gCodeErrorHandler(pMessage:=CONCAT('null reference in ',lIdentity));
END_IF

lRequestedRunState.MergeOutput := FALSE;
lRequestedRunState.EnumType := cEnumTypeRunState;
lRequestedRunState.initializeValueObjectOp(OpSelf,'ReqRunStt','Requested run state','',cValueStyleConfigurable);

lTargetVoltage.Scaling := 10.0;
lTargetVoltage.Offset := 0;
lTargetVoltage.initializeValueObjectOp(OpSelf,'VoltageReq','Target voltage','',cValueStyleConfigurable);

lVoltage.Scaling := 0.1;
lVoltage.Offset := 0;
lVoltage.initializeValueObjectOp(OpSelf,'VoltageCurr','Measured voltage','',cValueStyleConfigurable);

lCurrent.Scaling := 0.1;
lCurrent.Offset := 0.0;
lCurrent.initializeValueObjectOp(OpSelf,'CurrentCurr','Measured current','',cValueStyleConfigurable);

lTemperature.Scaling := 1.0;
lTemperature.Offset := 0.0;
lTemperature.initializeValueObjectOp(OpSelf,'Temp','Measured temperature','',cValueStyleConfigurable);

lDiagnosticState.initializeValueObjectOp(OpSelf,'Diagnostic','Diagnostic state','',cValueStyleConfigurable);

lStatusInitialization.Index := 0;
lStatusInitialization.initializeValueObjectOp(OpSelf,'Status','If current status is initialized','',cValueStyleConfigurable);
lStatusInitialization.InputReference REF= lDiagnosticState.ValueReference;

lStatusWorking.Index := 1;
lStatusWorking.initializeValueObjectOp(OpSelf,'Working','If current status is working','',cValueStyleConfigurable);
lStatusWorking.InputReference REF= lDiagnosticState.ValueReference;

(*//lFaultHardware.Index := 2; 16#4
//lFaultFan.Index := 6;16#40
//lFaultHVIL.Index := 7;16#80
lAlarmSecondaryHardware.initializeStateOp(OpSelf,cACSecondaryHardware);
lAlarmSecondaryHardware.Life := 10;
lAlarmSecondaryHardware.Severity := cSeverityCritical;
lAlarmSecondaryHardware.Mask := 16#C4;
lAlarmSecondaryHardware.InputReference REF= lDiagnosticState.ValueReference;

//lFaultCANBus.Index := 3;16#8
lAlarmSecondaryCANBus.initializeStateOp(OpSelf,cACSecondaryCANBus);
lAlarmSecondaryCANBus.Life := 10;
lAlarmSecondaryCANBus.Severity := cSeverityCritical;
lAlarmSecondaryCANBus.Mask := 16#8;
lAlarmSecondaryCANBus.InputReference REF= lDiagnosticState.ValueReference;

//lFaultShutdown.Index := 5;16#20
lAlarmSecondaryShutdown.initializeStateOp(OpSelf,cACSecondaryShutdown);
lAlarmSecondaryShutdown.Life := 10;
lAlarmSecondaryShutdown.Severity := cSeverityCritical;
lAlarmSecondaryShutdown.Mask := 16#20;
lAlarmSecondaryShutdown.InputReference REF= lDiagnosticState.ValueReference;

//lWarningTemperature.Index := 8;16#100
//lFaultTemperature.Index := 9;16#200
lAlarmSecondaryTemperature.initializeStateOp(OpSelf,cACSecondaryTemperature);
lAlarmSecondaryTemperature.Life := 10;
lAlarmSecondaryTemperature.Severity := cSeverityWarning;
lAlarmSecondaryTemperature.Mask := 16#300;
lAlarmSecondaryTemperature.InputReference REF= lDiagnosticState.ValueReference;

//lFaultInputOverVoltage.Index := 10;// 16#400
//lFaultInputUnderVoltage.Index := 11;16#800
lAlarmSecondaryInputVoltage.initializeStateOp(OpSelf,cACSecondaryInputVoltage);
lAlarmSecondaryInputVoltage.Life := 10;
lAlarmSecondaryInputVoltage.Severity := cSeverityError;
lAlarmSecondaryInputVoltage.Mask := 16#C00;
lAlarmSecondaryInputVoltage.InputReference REF= lDiagnosticState.ValueReference;

//lFaultOutputOverVoltage.Index := 12;16#1000
//lFaultOutputUnderVoltage.Index := 13;16#2000
lAlarmSecondaryOutputVoltage.initializeStateOp(OpSelf,cACSecondaryOutputVoltage);
lAlarmSecondaryOutputVoltage.Life := 10;
lAlarmSecondaryOutputVoltage.Severity := cSeverityError;
lAlarmSecondaryOutputVoltage.Mask := 16#3000;
lAlarmSecondaryOutputVoltage.InputReference REF= lDiagnosticState.ValueReference;

//lFaultOverCurrent.Index := 14;16#4000
lAlarmSecondaryOverCurrent.initializeStateOp(OpSelf,cACSecondaryOverCurrent);
lAlarmSecondaryOverCurrent.Life := 10;
lAlarmSecondaryOverCurrent.Severity := cSeverityError;
lAlarmSecondaryOverCurrent.Mask := 16#4000;
foobar lAlarmSecondaryOverCurrent.InputReference REF= lDiagnosticState.ValueReference;*)

lAlarmSecondaryTemperature.initializeState(NopSelf,'',cACSecondaryTemperature);
lAlarmSecondaryTemperature.registerServer(lSecondaryPowerSupply.Modulation);

lCurrentRunState.EnumType := cEnumTypeRunState;
lCurrentRunState.initializeValueObject(NopSelf,'CurrRunStt','Current run state','',cValueStyleConfigurable);

SUPER^.initialize();
SubSystem := cSubsystemSecondary;

lAlarmCANOpenSlaveNotOperational.InitialSeverity := cSeverityNone;
lAlarmCANOpenSlaveNotOperational.SeverityWarningTimeout := T#250MS;
lAlarmCANOpenSlaveNotOperational.SeverityErrorTimeout := T#1S;
lAlarmCANOpenSlaveNotOperational.SeverityCriticalTimeout := T#5S;

lAlarmCANOpenSlaveAllowableUp.AllowableSystemState := cSystemStatePreparing;
lAlarmCANOpenSlaveAllowableUp.UpperSystemStateScope := cSystemStatePreparing;
lAlarmCANOpenSlaveAllowableUp.LowerSystemStateScope := cSystemStatePreparing;

lStartSystemStateScope := t_system_state.cSystemStatePreparing;
lOperationalSystemStateScopeLower := t_system_state.cSystemStateCharging;
lModulationSystemStateScope := t_system_state.cSystemStateCharging;

                
END_METHOD

METHOD operator
                  SUPER^.operator();

IF (NOT(lEnabled)) THEN
	lCurrentRunState.Override := TRUE;
	lCurrentRunState.OverrideValue := cRunStateStart;
	
	RETURN;
END_IF

IF ((lStatusInitialization.Value) AND
	(lStatusWorking.Value)) THEN
	lCurrentRunState.Value := cRunStateStart;
ELSE	
	lCurrentRunState.Value := cRunStateStop;
END_IF

IF (WORD_TO_BOOL(UINT_TO_WORD(lDiagnosticState.Value) AND 16#7FEC)) THEN
	lAlarmCANOpenSlaveNotify.triggerWithContext(UINT_TO_WORD(lDiagnosticState.Value));
END_IF

IF (WORD_TO_BOOL(UINT_TO_WORD(lDiagnosticState.Value) AND 16#100)) THEN
	lAlarmSecondaryTemperature.ThresholdPositive := cAvailabilityTemperatureWarning;
	lAlarmSecondaryTemperature.trigger(FALSE);
END_IF
IF (WORD_TO_BOOL(UINT_TO_WORD(lDiagnosticState.Value) AND 16#200)) THEN
	lAlarmSecondaryTemperature.ThresholdPositive := cAvailabilityTemperatureFault;
	lAlarmSecondaryTemperature.trigger(FALSE);
END_IF

                
END_METHOD

METHOD initializeSecondary
  VAR_INPUT
    secondary : REFERENCE TO SecondaryPowerSupply;
  END_VAR
                  lSecondaryPowerSupply ref= secondary;
                
END_METHOD

METHOD initializeSecondaryIO
  VAR_INPUT
    voltage : REFERENCE TO UINT;
    current : REFERENCE TO UINT;
    temperature : REFERENCE TO USINT;
    state : REFERENCE TO UINT;
    control : REFERENCE TO USINT;
    targetVoltage : REFERENCE TO USINT;
  END_VAR
                  lVoltage.InputReference REF= voltage;
lCurrent.InputReference REF= current;
lTemperature.InputReference REF= temperature;

lDiagnosticState.InputReference REF= state;

lRequestedRunState.OutputReference REF= control;
lTargetVoltage.OutputReference REF= targetVoltage;


                
END_METHOD

METHOD notOperational
                  
                
END_METHOD

PROPERTY Current : REAL
GET
                    Current := lCurrent.Value;

                  
END_GET
END_PROPERTY

PROPERTY CurrentRunState : t_run_state
GET
                    lCurrentRunState.operator();
CurrentRunState := lCurrentRunState.Value;
                  
END_GET
END_PROPERTY

PROPERTY RequestedRunState : t_run_state
GET
                    RequestedRunState := lRequestedRunState.Value;
                  
END_GET
SET
                    lRequestedRunState.Value := RequestedRunState;


                  
END_SET
END_PROPERTY

PROPERTY TargetVoltage : REAL
GET
                    TargetVoltage := lTargetVoltage.Value;
                  
END_GET
SET
                    lTargetVoltage.Value := TargetVoltage;
                  
END_SET
END_PROPERTY

PROPERTY Temperature : REAL
GET
                    Temperature := lTemperature.Value;

                  
END_GET
END_PROPERTY

PROPERTY Voltage : REAL
GET
                    Voltage := lVoltage.Value;

                  
END_GET
END_PROPERTY
END_FUNCTION_BLOCK

FUNCTION_BLOCK ControllerSlavePLC EXTENDS CANOpenSlave
  VAR CONSTANT
    cNMTDetectionPeriod : t_time := TIME#2s500ms;
  END_VAR
  VAR
    lAlarmCANOpenSlaveNoValidTransmissions : ReportableAlarmAllowableUp;
    lVREnableDetectionTPDO : ValueReferenceBool;
    lEnableDetectionTPDO : BOOL := TRUE;
    lVREnableValidTransmissions : ValueReferenceBool;
    lEnableValidTransmissions : BOOL := FALSE;
    lEnableNMTDetectionTPDO : BOOL := FALSE;
    lEnableNMTOverrideTPDO : BOOL := TRUE;
    lNMTDetectionTimer : t_timer;
    lTPDO1Stuffing : BOOL;
    lTPDO1StuffingPrevious : BOOL;
  END_VAR

            ;
          

METHOD initialize
                  lVREnableDetectionTPDO.initializeValueReference(lEnableDetectionTPDO,NopSelf,'EnblDtctTPDO','Use TPDO traffic to determine node state','',cValueStyleParameter);
lVREnableValidTransmissions.initializeValueReference(lEnableValidTransmissions,NopSelf,'EnblVldTrnms','Check if TPDO traffic is valid','',cValueStyleParameter);
	
lAlarmCANOpenSlaveNoValidTransmissions.initializeState(NopSelf,'',cACCANOpenSlaveNoValidTransmissions);
lAlarmCANOpenSlaveNoValidTransmissions.AllowableSystemState := cSystemStatePreparing;
lAlarmCANOpenSlaveNoValidTransmissions.UpperSystemStateScope := cSystemStatePreparing;
lAlarmCANOpenSlaveNoValidTransmissions.LowerSystemStateScope := cSystemStatePreparing;
lAlarmCANOpenSlaveNoValidTransmissions.Life := 10;
lAlarmCANOpenSlaveNoValidTransmissions.InitialSeverity := cSeverityNone;
lAlarmCANOpenSlaveNoValidTransmissions.SeverityWarningTimeout := T#2S;
lAlarmCANOpenSlaveNoValidTransmissions.SeverityErrorTimeout := T#4S;
lAlarmCANOpenSlaveNoValidTransmissions.SeverityCriticalTimeout := T#10S;	

SUPER^.initialize();

lNMTDetectionTimer.initialize();
lNMTDetectionTimer.Enable := TRUE;
lNMTDetectionTimer.Period := cNMTDetectionPeriod;
                
END_METHOD

METHOD operator
                  SUPER^.operator();

lTPDO1StuffingPrevious := lTPDO1Stuffing;
lTPDO1Stuffing := Peripheral.TPDO1Stuffing;

IF (NOT(ValidTransmissions)) THEN
	lAlarmCANOpenSlaveNoValidTransmissions.test(FALSE);
END_IF




                
END_METHOD

PROPERTY NodeState : t_node_state
SET
                    IF (lEnableDetectionTPDO) THEN

	IF (lTPDO1StuffingPrevious<>lTPDO1Stuffing) THEN
		lNMTDetectionTimer.reset();
	END_IF
	
	lNMTDetectionTimer.operator();
	IF (NOT(lNMTDetectionTimer.Expired)) THEN
		lNodeState := NodeState;
		
		IF (lEnableNMTDetectionTPDO) THEN
			lNodeState := t_node_state.OPERATIONAL;
		END_IF

		RETURN;
	END_IF

	IF (lEnableNMTOverrideTPDO) THEN
		lNodeState := t_node_state.NOT_AVAIL;
		RETURN;
	END_IF	
END_IF

lNodeState := NodeState;

                  
END_SET
END_PROPERTY

PROPERTY Peripheral : REFERENCE TO Peripheral
GET
                    
                  
END_GET
END_PROPERTY

PROPERTY ValidTransmissions : BOOL
GET
                    IF (NOT(lEnableValidTransmissions)) THEN
	ValidTransmissions := TRUE;
	RETURN;
END_IF

ValidTransmissions := ((NodeState=t_node_state.OPERATIONAL) AND
	(Peripheral.ValidTransmissions));

                  
END_GET
END_PROPERTY
END_FUNCTION_BLOCK

FUNCTION_BLOCK SecondaryPowerSupply EXTENDS NonOperationalParticleSet
  VAR CONSTANT
    cSecondaryTargetVoltage : REAL := 13.0;
    cStartDelayPeriod : t_time := TIME#1s0ms;
  END_VAR
  VAR
    lAlarmSecondaryWaiting : ReportableAlarmAllowableUp;
    lAlarmSecondaryNotRunning : ReportableAlarmEscalating;
    lAlarmSecondaryNotRunningModulation : ReportableSignedModulation;
    lAlarmRunStateMismatch : ReportableAlarmEscalating;
    lModulation : ReportableContextSignedModulation;
    lAvailability : t_percentage;
    lModulationSeverity : t_severity;
    lRequestedState : t_run_state;
    lCurrentState : t_run_state;
    lTargetVoltage : REAL;
    lControllerSecondaryPowerSupplyA : REFERENCE TO ControllerSecondaryPowerSupply;
    lControllerSecondaryPowerSupplyB : REFERENCE TO ControllerSecondaryPowerSupply;
    lStartDelayTimer : t_timer;
  END_VAR

            ;
          

METHOD initialize
                  IF ((NOT(__ISVALIDREF(lControllerSecondaryPowerSupplyA))) OR
	(NOT(__ISVALIDREF(lControllerSecondaryPowerSupplyB)))) THEN
	gCodeErrorHandler(pMessage:=CONCAT('null reference in ',lIdentity));
END_IF

lAlarmSecondaryNotRunning.initializeState(NopSelf,'',cACSecondaryNotRunning); // foobar escalates to pause
lAlarmSecondaryNotRunning.Life := 10;
lAlarmSecondaryNotRunning.InitialSeverity := cSeverityNone;
lAlarmSecondaryNotRunning.SeverityWarningTimeout := T#1S;
lAlarmSecondaryNotRunning.SeverityErrorTimeout := T#2S;
lAlarmSecondaryNotRunning.SeverityCriticalTimeout := T#5S;

lAlarmSecondaryNotRunningModulation.initializeState(NopSelf,'',cACSecondaryNotRunningModulation); // foobar life was zero
lAlarmSecondaryNotRunningModulation.pause();
lAlarmSecondaryNotRunningModulation.registerServer(ADR(lModulation));

lAlarmSecondaryWaiting.initializeState(NopSelf,'',cACSecondaryWaiting);
lAlarmSecondaryWaiting.AllowableSystemState := cSystemStatePreparing;
lAlarmSecondaryWaiting.UpperSystemStateScope := cSystemStatePreparing;
lAlarmSecondaryWaiting.LowerSystemStateScope := cSystemStatePreparing;
lAlarmSecondaryWaiting.Life := 10;
lAlarmSecondaryWaiting.InitialSeverity := cSeverityNone;
lAlarmSecondaryWaiting.SeverityWarningTimeout := T#1S;
lAlarmSecondaryWaiting.SeverityErrorTimeout := T#2S;
lAlarmSecondaryWaiting.SeverityCriticalTimeout := T#5S;

lAlarmRunStateMismatch.initializeState(NopSelf,'',cACSecondaryRunStateMismatch);
lAlarmRunStateMismatch.InitialSeverity := cSeverityNone;
lAlarmRunStateMismatch.SeverityWarningTimeout := T#2S;
lAlarmRunStateMismatch.SeverityErrorTimeout := T#4S;
lAlarmRunStateMismatch.SeverityCriticalTimeout := T#6S;

lModulation.initializeEvent(NopSelf,'',cECSecondaryPowerModulation);

SUPER^.initialize();
SubSystem := cSubsystemSecondary;

lModulationSeverity := cSeverityError;
lTargetVoltage := cSecondaryTargetVoltage;

lStartDelayTimer.Enable := TRUE;
lStartDelayTimer.Period := cStartDelayPeriod;
lStartDelayTimer.initialize();
                
END_METHOD

METHOD operator
                  lCurrentState := cRunStateNone;

IF ((lControllerSecondaryPowerSupplyA.CurrentRunState=cRunStateStop) OR
	(lControllerSecondaryPowerSupplyB.CurrentRunState=cRunStateStop)) THEN
	lCurrentState := cRunStateStop;
END_IF

IF ((lControllerSecondaryPowerSupplyA.CurrentRunState=cRunStateStart) AND
	(lControllerSecondaryPowerSupplyB.CurrentRunState=cRunStateStart)) THEN
	lCurrentState := cRunStateStart;
END_IF
	
IF (lControllerSecondaryPowerSupplyA.CurrentRunState<>lControllerSecondaryPowerSupplyB.CurrentRunState) THEN
	lAlarmRunStateMismatch.trigger(FALSE); // foobar any further action
END_IF

SUPER^.operator();

lRequestedState := cRunStateStop;
lAvailability := 0.0;

IF (gSystemServices.SystemState.State<cSystemStatePreparing) THEN
	RETURN;
END_IF

IF (BMSConnected) THEN
	lRequestedState := cRunStateStart;
ELSE
	lStartDelayTimer.reset();	
END_IF
lStartDelayTimer.operator();

IF (lCurrentState<>cRunStateStart) THEN
	lAlarmSecondaryNotRunning.trigger(FALSE);
	
	IF (lAlarmSecondaryNotRunning.Severity>=lModulationSeverity) THEN
		lAlarmSecondaryNotRunningModulation.trigger(FALSE);
	END_IF

	lAlarmSecondaryWaiting.test(FALSE);	
END_IF

lModulation.operator();
lAvailability := MIN(lModulation.ScalingPositive,lModulation.ThresholdPositive);

lControllerSecondaryPowerSupplyA.RequestedRunState := lRequestedState;
IF ((lStartDelayTimer.Expired) AND (lRequestedState=cRunStateStart)) THEN
	lControllerSecondaryPowerSupplyB.RequestedRunState := cRunStateStart;
ELSE
	lControllerSecondaryPowerSupplyB.RequestedRunState := cRunStateStop;	
END_IF

lControllerSecondaryPowerSupplyA.TargetVoltage := lTargetVoltage;
lControllerSecondaryPowerSupplyB.TargetVoltage := lTargetVoltage;

                
END_METHOD

PROPERTY Availability : t_percentage
GET
                    Availability := lAvailability;
                  
END_GET
END_PROPERTY

PROPERTY CurrentState : t_run_state
GET
                    CurrentState := lCurrentState;

                  
END_GET
END_PROPERTY

PROPERTY Modulation : POINTER TO ReportableContextSignedModulation
GET
                    Modulation := ADR(lModulation);

                  
END_GET
END_PROPERTY

PROPERTY RequestedState : t_run_state
GET
                    RequestedState := lRequestedState;

                  
END_GET
END_PROPERTY

PROPERTY Running : BOOL
GET
                    Running := (lCurrentState=cRunStateStart);

                  
END_GET
END_PROPERTY

PROPERTY TargetVoltage : REAL
GET
                    TargetVoltage := lTargetVoltage;
                  
END_GET
SET
                    lTargetVoltage := TargetVoltage;
                  
END_SET
END_PROPERTY

PROPERTY TypeToken : t_medium_string
GET
                    TypeToken := 'Secondary';
                  
END_GET
END_PROPERTY

PROPERTY BMSConnected : BOOL
GET
                    BMSConnected := false;
                  
END_GET
END_PROPERTY
END_FUNCTION_BLOCK

FUNCTION_BLOCK SecondaryPowerSupplyPrimary EXTENDS SecondaryPowerSupply

            ;
          

METHOD initialize
                  SUPER^.initialize();

lControllerSecondaryPowerSupplyA REF= gSystem.lCANOpenMasterSystem.SecondaryPowerSupplyA;
lControllerSecondaryPowerSupplyB REF= gSystem.lCANOpenMasterSystem.SecondaryPowerSupplyB;

                
END_METHOD
END_FUNCTION_BLOCK
